FUNCTION BYTE2n08b
  (* Standard: 61499-1 *)
  (* Version 1.0, 2024-02-22, franz *)
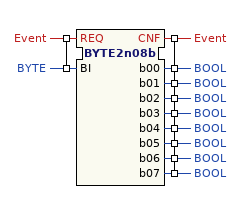
  EVENT_INPUT
    REQ WITH BI;
  END_EVENT
  EVENT_OUTPUT
    CNF WITH b00, b01, b02, b03, b04, b05, b06, b07;
  END_EVENT
  VAR_INPUT
    BI : BYTE;
  END_VAR
  VAR_OUTPUT
    b00 : BOOL; (* BIT 00 *)
    b01 : BOOL; (* BIT 01 *)
    b02 : BOOL; (* BIT 02 *)
    b03 : BOOL; (* BIT 03 *)
    b04 : BOOL; (* BIT 04 *)
    b05 : BOOL; (* BIT 05 *)
    b06 : BOOL; (* BIT 06 *)
    b07 : BOOL; (* BIT 07 *)
  END_VAR
  BODY IN ST:
FUNCTION BYTE2n08b

VAR_INPUT
	BI : BYTE;
END_VAR

VAR_OUTPUT
	b00 : BOOL;    // BIT 00
	b01 : BOOL;    // BIT 01
	b02 : BOOL;    // BIT 02
	b03 : BOOL;    // BIT 03
	b04 : BOOL;    // BIT 04
	b05 : BOOL;    // BIT 05
	b06 : BOOL;    // BIT 06
	b07 : BOOL;    // BIT 07
END_VAR

END_FUNCTION
  END_BODY
END_FUNCTION
